// Mitsubishi GX Works2 project: counter+sequence_2   PLC: Q03UDV

PROGRAM MAIN
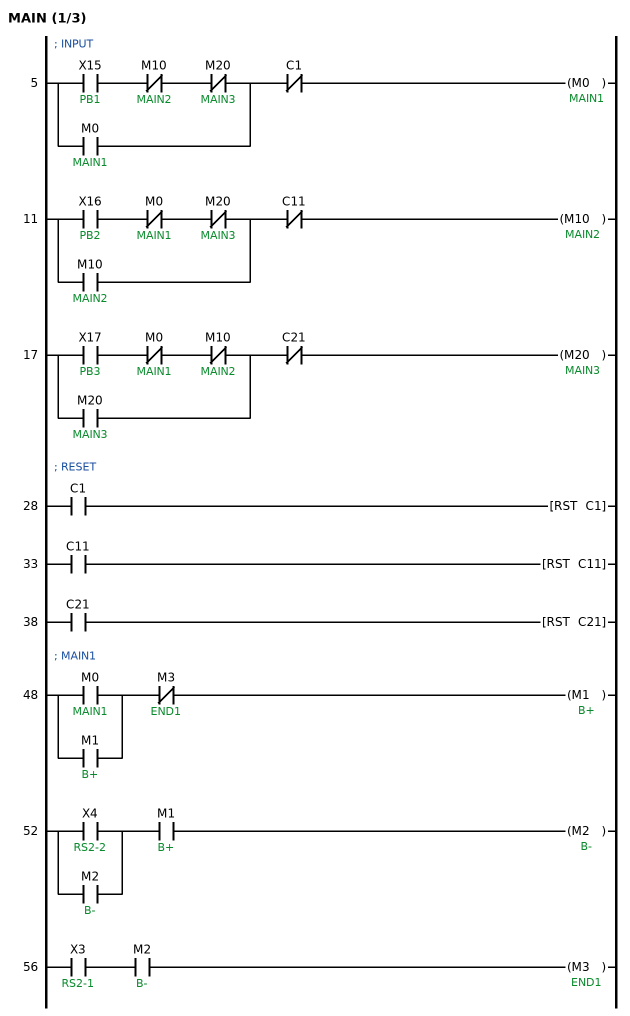
; INPUT
5     LD      X15  ; PB1
      ANI     M10  ; MAIN2
      ANI     M20  ; MAIN3
      OR      M0  ; MAIN1
      ANI     C1
      OUT     M0  ; MAIN1
11    LD      X16  ; PB2
      ANI     M0  ; MAIN1
      ANI     M20  ; MAIN3
      OR      M10  ; MAIN2
      ANI     C11
      OUT     M10  ; MAIN2
17    LD      X17  ; PB3
      ANI     M0  ; MAIN1
      ANI     M10  ; MAIN2
      OR      M20  ; MAIN3
      ANI     C21
      OUT     M20  ; MAIN3
; RESET
28    LD      C1
      RST     C1
33    LD      C11
      RST     C11
38    LD      C21
      RST     C21
; MAIN1
48    LD      M0  ; MAIN1
      OR      M1  ; B+
      ANI     M3  ; END1
      OUT     M1  ; B+
52    LD      X4  ; RS2-2
      OR      M2  ; B-
      AND     M1  ; B+
      OUT     M2  ; B-
56    LD      X3  ; RS2-1
      AND     M2  ; B-
      OUT     M3  ; END1
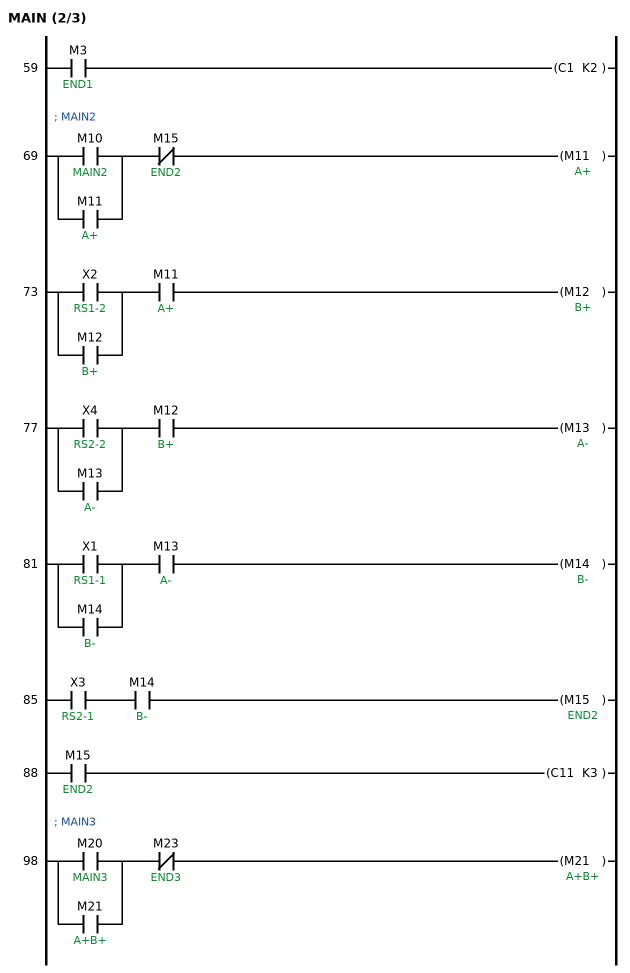
59    LD      M3  ; END1
      OUT     C1 K2
; MAIN2
69    LD      M10  ; MAIN2
      OR      M11  ; A+
      ANI     M15  ; END2
      OUT     M11  ; A+
73    LD      X2  ; RS1-2
      OR      M12  ; B+
      AND     M11  ; A+
      OUT     M12  ; B+
77    LD      X4  ; RS2-2
      OR      M13  ; A-
      AND     M12  ; B+
      OUT     M13  ; A-
81    LD      X1  ; RS1-1
      OR      M14  ; B-
      AND     M13  ; A-
      OUT     M14  ; B-
85    LD      X3  ; RS2-1
      AND     M14  ; B-
      OUT     M15  ; END2
88    LD      M15  ; END2
      OUT     C11 K3
; MAIN3
98    LD      M20  ; MAIN3
      OR      M21  ; A+B+
      ANI     M23  ; END3
      OUT     M21  ; A+B+
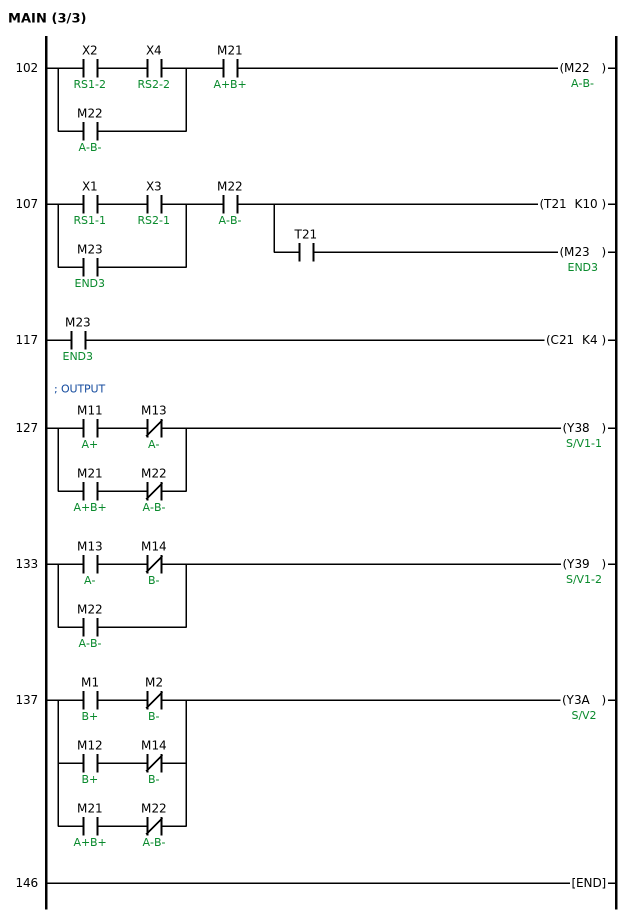
102   LD      X2  ; RS1-2
      AND     X4  ; RS2-2
      OR      M22  ; A-B-
      AND     M21  ; A+B+
      OUT     M22  ; A-B-
107   LD      X1  ; RS1-1
      AND     X3  ; RS2-1
      OR      M23  ; END3
      AND     M22  ; A-B-
      OUT     T21 K10
      AND     T21
      OUT     M23  ; END3
117   LD      M23  ; END3
      OUT     C21 K4
; OUTPUT
127   LD      M11  ; A+
      ANI     M13  ; A-
      LD      M21  ; A+B+
      ANI     M22  ; A-B-
      ORB
      OUT     Y38  ; S/V1-1
133   LD      M13  ; A-
      ANI     M14  ; B-
      OR      M22  ; A-B-
      OUT     Y39  ; S/V1-2
137   LD      M1  ; B+
      ANI     M2  ; B-
      LD      M12  ; B+
      ANI     M14  ; B-
      ORB
      LD      M21  ; A+B+
      ANI     M22  ; A-B-
      ORB
      OUT     Y3A  ; S/V2
146   END
END_PROGRAM

// device comments not shown above
X18  ; PB4
X1B  ; PB7
M4  ; B-
M31  ; B+
M32  ; B-A+
M33  ; A-
